{attribute 'linkalways'} 
{attribute 'no_explicit_call' := 'This FB is a CLASS and must be accessed using methods or properties'}
{attribute 'enable_dynamic_creation'}
FUNCTION_BLOCK FINAL SEL_DWORD EXTENDS Node
VAR
	g : _BOOL(FALSE);
	in1 : _DWORD(0);
	in2 : _DWORD(0);
	out : _DWORD(0);
END_VAR

METHOD PUBLIC Clone : I_Node
VAR
	pNode : POINTER TO SEL_DWORD;
END_VAR
pNode := __NEW(SEL_DWORD);
Clone := pNode^;
END_METHOD

METHOD FB_init : BOOL
VAR_INPUT
	bInitRetains : BOOL; // if TRUE, the retain variables are initialized (warm start / cold start)
	bInCopyCode : BOOL;  // if TRUE, the instance afterwards gets moved into the copy code (online change)
END_VAR
AddInput('g',THIS^.g);
AddInput('in1',THIS^.in1);
AddInput('in2',THIS^.in2);
AddOutput('out', THIS^.out);
END_METHOD

METHOD PROTECTED OnExecute
VAR
END_VAR
IF g.value THEN
	out.value := in2.value;
ELSE
	out.value := in1.value;
END_IF
END_METHOD

END_FUNCTION_BLOCK

(* stored: Version 1.1.0.1, ProductVersion 3.1.4024.15
   POU SEL_DWORD: Id {5f9e6364-123d-47a7-afb6-f1b7b2d673ad}, SpecialFunc None
   Folder Constructor: Id {307c42b3-de0c-4787-8487-b23bd231ccc8}
   Method Clone: Id {75cc739b-4101-49c6-a866-1788c26cc476}
   Method FB_init: Id {f0859ac3-edcf-42cd-ab71-b4aa74542cd9}
   Method OnExecute: Id {d0b0fe9e-2c4e-49ba-8065-3a0ca16d599c} *)
